Staubli VAL3: refreshStatic.pgx

program refreshStatic()
  local string l_sMenu
  local string l_sMessage
  local string l_sMotorStatus
begin
  cls()
  //
  // set the view of the page..
  //
  // SET THE PAGE NUMBER
  use:nPage=110
  // load the menu page

  l_sMessage=" -,test,复位,,,, +,"

  // define the menu
  call use:stringToArray(l_sMessage,sMenu)
  call use:setMenu(sMenu,true,3)
  call use:getMenu(sMenu,bButton)
  //
  // CREATE THE LIST
  //
  // define your list size for default
  call use:setSizeList(21,0,17,10)
  // set small nParView
  call use:setView(false)
  //
  call use:listcreate("AXIS8 ")
  //
  call use:listadd(sList)
  //
  // refresh the cursor
  // select the last item
  call use:selectNewField(nSelected,nIndex,nView)


  if aioGet(MbAI_b8MotorErr)==1
    l_sMotorStatus=l_sMotorStatus+" 马达错误"
  else
    l_sMotorStatus=l_sMotorStatus+" 马达正常"
  endIf

  call use:type(0,1,l_sMotorStatus)

end
